FUNCTION_BLOCK Q_ListItem (* Command change list item ( Part 6 - F.42 ) *)
  (* Standard: ISO 11783-6; Description: Copyright (c) 2022 HR Agrartechnik GmbH This program and the accompanying materials are made available under the terms of the Eclipse Public License 2.0 which is available at https://www.eclipse.org/legal/epl-2.0/ SPDX-License-Identifier: EPL-2.0 see Description Tab *)
  (* Version 1.0, 2022-07-08, Franz Höpfinger, HR Agrartechnik GmbH *)
  (* Documentation:
  Command change list item ( Part 6 - F.42 )
   This command is used to change a list item in a list input object.
   param[in] {objectID, uint16_t}
   Object ID of a list input object
   param[in] {listIndex, uint8_t}
   List index (-> see list)
   param[in] {newObjectID, uint16_t}
   New object ID or 0xFFFF to set empty
   Return Values: 
   int16_t
    - VT_E_NO_ERR (0) - OK
   - VT_E_OVERFLOW (-6) - buffer overflow
   - VT_E_NOACT (-8) - Command not possible in current state
   - VT_E_NO_INSTANCE (-21) - No VT client available
   - VT_E_ISO_INSTANCE_INVALID (-129) - Identifier for instance (connection) invalid
   - VT_E_NOT_ALIVE (-130) - Identifier for instance valid, but VT Dead.
  *)
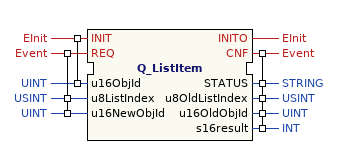
  EVENT_INPUT
    INIT : EInit WITH u16ObjId; (* Service Initialization *)
    REQ WITH u8ListIndex, u16NewObjId; (* Service Request *)
  END_EVENT
  EVENT_OUTPUT
    INITO : EInit; (* Initialization Confirm *)
    CNF WITH STATUS, s16result, u8OldListIndex, u16OldObjId; (* Confirmation of Requested Service *)
  END_EVENT
  VAR_INPUT
    u16ObjId : UINT; (* Object ID *)
    u8ListIndex : USINT; (* List index (-> see list) *)
    u16NewObjId : UINT; (* New object ID or 0xFFFF to set empty *)
  END_VAR
  VAR_OUTPUT
    STATUS : STRING; (* Service Status *)
    u8OldListIndex : USINT; (* Old list index (-> see list) *)
    u16OldObjId : UINT; (* Old object ID or 0xFFFF to set empty *)
    s16result : INT; (* retval see description *)
  END_VAR
END_FUNCTION_BLOCK
